// SIMATIC S7-200 project (STEP 7-Micro/WIN), CPU 224XP REL 02.01

ORGANIZATION_BLOCK Bloque_de_programa:OB1
TITLE=COMENTARIOS DEL PROGRAMA
BEGIN
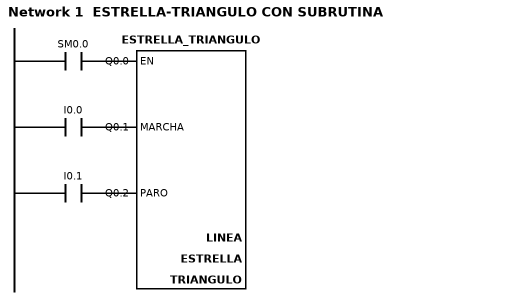
Network 1 // ESTRELLA-TRIANGULO CON SUBRUTINA
// (network saved uncompiled; LAD cells follow)
// row 0: c0 -| |- SM0.0  c1 [ESTRELLA_TRIANGULO LINEA ESTRELLA TRIANGULO EN:=Q0.0, MARCHA:=Q0.1, PARO:=Q0.2]
// row 1: c0 -| |- I0.0  c1 [box]
// row 2: c0 -| |- I0.1  c1 [box]
// row 3: c1 [box]
END_ORGANIZATION_BLOCK

SUBROUTINE_BLOCK ESTRELLA_TRIANGULO:SBR0
TITLE=COMENTARIOS DE LA SUBRUTINA
VAR_INPUT
MARCHA:BOOL;	// L0.0 
PARO:BOOL;	// L0.1 
END_VAR
VAR_OUTPUT
LINEA:BOOL;	// L0.2 
ESTRELLA:BOOL;	// L0.3 
TRIANGULO:BOOL;	// L0.4 
END_VAR
BEGIN
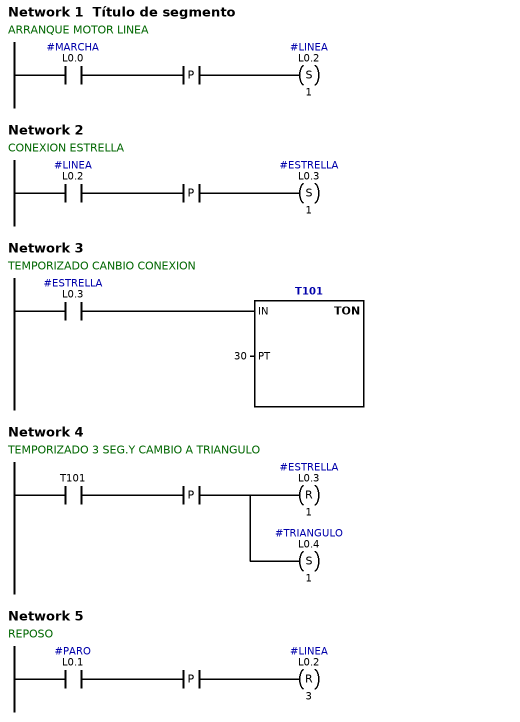
Network 1 // Título de segmento
// ARRANQUE MOTOR LINEA
// (network saved uncompiled; LAD cells follow)
// row 0: c0 -| |- #MARCHA:L0.0  c1 -|P|-  c2 -(S) #LINEA:L0.2, 1
Network 2
// CONEXION ESTRELLA
// (network saved uncompiled; LAD cells follow)
// row 0: c0 -| |- #LINEA:L0.2  c1 -|P|-  c2 -(S) #ESTRELLA:L0.3, 1
Network 3
// TEMPORIZADO CANBIO CONEXION
// (network saved uncompiled; LAD cells follow)
// row 0: c0 -| |- #ESTRELLA:L0.3  c1 --  c2 [TON T101 IN:=power@row0, PT:=30]
// row 1: c2 [box]
Network 4
// TEMPORIZADO 3 SEG.Y CAMBIO A TRIANGULO
// (network saved uncompiled; LAD cells follow)
// row 0: c0 -| |- T101  c1 -|P|-  v  c2 -(R) #ESTRELLA:L0.3, 1
// row 1: c1 ^  c2 -(S) #TRIANGULO:L0.4, 1
Network 5
// REPOSO
// (network saved uncompiled; LAD cells follow)
// row 0: c0 -| |- #PARO:L0.1  c1 -|P|-  c2 -(R) #LINEA:L0.2, 3
END_SUBROUTINE_BLOCK
